FUNCTION_BLOCK E_SPLIT_3 (* Based on E_SPLIT with 3 outputs *)
  (* Standard: 61499-2 *)
  (* Version 1.0, 2017-06-07, Marc Jakobi, HTW Berlin *)
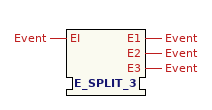
  EVENT_INPUT
    EI; (* Input event *)
  END_EVENT
  EVENT_OUTPUT
    E1; (* Execution Confirmation *)
    E2;
    E3;
  END_EVENT
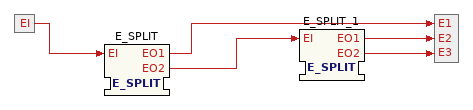
  FBS
    E_SPLIT : E_SPLIT;
    E_SPLIT_1 : E_SPLIT;
  END_FBS
  EVENT_CONNECTIONS
    EI TO E_SPLIT.EI;
    E_SPLIT.EO1 TO E1;
    E_SPLIT.EO2 TO E_SPLIT_1.EI;
    E_SPLIT_1.EO1 TO E2;
    E_SPLIT_1.EO2 TO E3;
  END_CONNECTIONS
END_FUNCTION_BLOCK
